# EPICS substitutions: PIP-II/RFPI2/rfpi-fdr-sw-mgmt-ioc-main/ina-managementApp/Db/circuit.substitutions
file shortopen.template {
pattern{ acc, sys, group, num }
{ PIP2IT, pHB650, RFPI, CS0 }
{ PIP2IT, pHB650, RFPI, CS1 }
{ PIP2IT, pHB650, RFPI, SSA }
}
